Staubli VAL3: page.pgx

public program page(string& menuname[], num index)
// set all the page in english
begin
  //
  //  PAGE
  //
  //
  // PALLET PAGE
  if index>=10 and index<=19
    title("<货盘页面>")
  endIf
  // PALLET VIEW PAGE
  if index>=100 and index<=109
    title("<货盘浏览>")
  endIf
  switch index
    //
    // PALLET
    //
    // Integrator programmer
    case 10,11
      menuname="浏览,编辑,,,向导,复位,返回,继续"
    break
    // On Cycle
    case 13,14
      menuname="浏览,编辑,,,,复位,返回,继续"
    break
    // VIEW PALLET
    case 100,101,102,103,104,105
      menuname="复位全部,,,,,复位,返回,继续"
    break
  endSwitch
end
